PROGRAM PRG_PLC1
VAR
	EncoderValue AT %I* : UINT;
	Pos					: LREAL;
	ProcessingTime		:UDINT:=50;
END_VAR

F_ConsumeTime(ProcessingTime);

Pos:= UINT_TO_LREAL(EncoderValue)*100;

END_PROGRAM

(* stored: Version 1.1.0.1, ProductVersion 3.1.4026.18
   POU PRG_PLC1: Id {99e8ecb6-2e62-43ad-aace-946c2769ef26}, SpecialFunc None *)
